// TwinCAT 3 PLC project Tc_PidControl
// ProgramVersion: 3.1.4024.0
// libraries:
//   PlantControl and CMs, * (ArmAutomation)
//   Tc2_ControllerToolbox, * (Beckhoff Automation GmbH)
//   Tc2_Standard, * (Beckhoff Automation GmbH)
//   Tc2_System, * (Beckhoff Automation GmbH)
//   Tc3_Module, * (Beckhoff Automation GmbH)
// project tree:
//   / CyclicTask100Ms.TcTTO, PlcTask.TcTTO
//   DUTs/ stParamsForScaling.TcDUT
//   GVLs/ FIO.TcGVL, GVL.TcGVL, IO.TcGVL
//   POUs/ MAIN.TcPOU
//   POUs/PID/ PRG_FB_CTRL_EmptyTank.TcPOU, PRG_FB_CTRL_PID.TcPOU, PRG_PID_CALL.TcPOU
//   POUs/Scaling/ FB_ScaleIN.TcPOU (not stored), FB_ScaleOut.TcPOU
// real-time tasks:
//   TASK PlcTask: cycle T#10ms, priority 20, ADS port 350
//   TASK CyclicTask100Ms: cycle T#100000us, priority 1, ADS port 351
// I/O:
//   DEVICE Device 1 (EtherCAT) (disabled), AmsNetId 192.168.0.244.2.1
//     Term 1 (EK1200) [EK1200-5000 EtherCAT Power supply (2A E-Bus)]
//       Term 2 (EL1008) [EL1008 8Ch. Dig. Input 24V, 3ms]
//       Term 3 (EL2008) [EL2008 8Ch. Dig. Output 24V, 0.5A]
//       Term 4 (EL3044) [EL3044 4Ch. Ana. Input 0-20mA]
//       Term 5 (EL3174) [EL3174 4Ch. Ana. Input +/-10V Diff., +/-20mA SingleEnded, 16 Bit]
//       Term 6 (EL4014) [EL4014 4Ch. Ana. Output 0-20mA, 12bit]
// variable links:
//   Tc_PidControl/Tc_PidControl Instance <-> Device 1 (EtherCAT)/Term 1 (EK1200)/Term 5 (EL3174)
//     PlcTask Inputs/IO.aiSpare02c <-> AI Standard Channel 3/Value
//     PlcTask Inputs/IO.aiSpare02d <-> AI Standard Channel 4/Value

CONFIGURATION Tc_PidControl
    RESOURCE PLC ON TwinCAT3
        TASK CyclicTask100Ms(INTERVAL := T#100000us, PRIORITY := 1);
        TASK PlcTask(INTERVAL := T#10ms, PRIORITY := 20);
        PROGRAM PRG_PID_CALL WITH CyclicTask100Ms : PRG_PID_CALL;
        PROGRAM MAIN WITH PlcTask : MAIN;
    END_RESOURCE
END_CONFIGURATION

// ---- DUTs/stParamsForScaling.TcDUT
TYPE stParamsForScaling :
STRUCT
	
    tCtrlCycleTime  : TIME := T#0ms; 
    tTaskCycleTime  : TIME := T#0ms; 
    fInMin          : REAL;
    fInMax          : REAL;
    fOutMin         : REAL;
    fOutMax         : REAL;
	
END_STRUCT

END_TYPE

// ---- GVLs/FIO.TcGVL
{attribute 'qualified_only'}
VAR_GLOBAL
	
	//	Sensor/Actuator	 Data TYPE	 Name	 Address	 Current Value
	//	Sensor	BOOL	FACTORY I/O (Running)	496	FALSE
	//	Sensor	Bool	FACTORY I/O (Paused)	497	FALSE
	//	Sensor	Bool	FACTORY I/O (Reset)	498	FALSE
	//bStart : BOOL;//	Sensor	Bool	Start	0	FALSE
	//bStop : BOOL;//	Sensor	Bool	Stop	1	TRUE
	//bReset : BOOL;//	Sensor	Bool	Reset	2	FALSE
	//	Sensor	Float	FACTORY I/O (Time Scale)	240	0
	rFlowMeter : REAL;	//	Sensor	Float	Flow meter	1	0
	rLevelMeter : REAL;	//	Sensor	Float	Level meter	0	0
	rSetPoint : REAL;	//	Sensor	Float	Setpoint	2	0
	rDisturbanceInput : REAL;
	rDisturbanceDisplay : DINT;
	//	Actuator	Bool	FACTORY I/O (Run)	496	FALSE
	//	Actuator	Bool	FACTORY I/O (Pause)	497	FALSE
	//	Actuator	Bool	FACTORY I/O (Reset)	498	FALSE
	//	Actuator	Bool	Start light	0	FALSE
	//	Actuator	Bool	Stop light	1	FALSE
	//	Actuator	Bool	Reset light	2	FALSE
	rDischargeValve : REAL;//	Actuator	Float	Discharge valve	1	0
	rFillValve : REAL;//	Actuator	Float	Fill valve	0	0
	//	Actuator	Int	FACTORY I/O (Camera Position)	240	0
	iSP : DINT;//	Actuator	Int	SP	0	0
	iPV : DINT;//	Actuator	Int	PV	1	0

END_VAR

// ---- GVLs/GVL.TcGVL
{attribute 'qualified_only'}
VAR_GLOBAL
	rAIInput1 : REAL;
	rAIInput2 : REAL;
	
	fSetpointValueToScope : LREAL;
	fActualValueToScope : LREAL;
	foutToScope : LREAL;
	
	outputDischargeValve : REAL;
	scaledDisturbancePotmeter : REAL;
	
	StartStep5 : BOOL;
	StartStep10 : BOOL;
	StartStep15 : BOOL;
	
	setManual : BOOL;
	setAuto : BOOL;
	
END_VAR

// ---- GVLs/IO.TcGVL
{attribute 'qualified_only'}
VAR_GLOBAL
	
	//EL3044
	aiSpare01a AT %I*: INT;
	aiSpare01b AT %I*: INT;
	aiSpare01c AT %I*: INT;
	aiSpare01d AT %I*: INT;
	
	//EL3074
	aiSpare02a AT %I*: INT;
	aiSpare02b AT %I*: INT;
	aiSpare02c AT %I*: INT; //ch3 0-10v  Legacy range			(0-32767)
	aiSpare02d AT %I*: INT; //ch4 0-20mA Extended range 		(0 -30518)
	
END_VAR

// ---- POUs/PID/PRG_PID_CALL.TcPOU
PROGRAM PRG_PID_CALL
VAR
	fbPlantControl : PlantAndCMs.FB_PlantControl_mode_2;
	Udt_FbPlantControl : PlantAndCMs.Udt_PlantControl_Mode_2;
	
	fbScalingSetpoint : FB_ScaleIN;
	fbScalingLevelMeter : FB_ScaleIN;
END_VAR


PRG_FB_CTRL_PID();
PRG_FB_CTRL_EmptyTank();


fbScalingSetpoint(
	taskCycletime := T#100MS,
	ctrlCycletime := T#100MS,
	inMin := 0.0,
	inMax := 10.0,
	outMin := 0.0,
	outMax := 300,
	
	inputForScaling := FIO.rSetPoint,
	
	scaledOutputInt => FIO.iSP
	);
fbScalingLevelMeter(
	taskCycletime := T#100MS,
	ctrlCycletime := T#100MS,
	inMin := 0.0,
	inMax := 10.0,
	outMin := 0.0,
	outMax := 300,
	
	inputForScaling := FIO.rLevelMeter,
	
	scaledOutputInt => FIO.iPV
	);


//aiSpare02c AT %I*: INT; //ch3 0-10v  Legacy range			(0-32767)
//measure 0-10v
//GVL.rAIInput1 := (INT_TO_REAL(IO.aiSpare02c)/(32767.0-0.0)) * 10.0;

//aiSpare02d AT %I*: INT; //ch4 0-20mA Extended range 		(0 -30518)
//measure 0-100%
//GVL.rAIInput2 := (INT_TO_REAL(IO.aiSpare02d)/(30518.0-0.0)) * 100.0;

END_PROGRAM

// ---- POUs/PID/PRG_FB_CTRL_PID.TcPOU
PROGRAM PRG_FB_CTRL_PID
VAR
	fSetpointValue					: LREAL;
	fActualValue					: LREAL;
	fManSyncValue					: LREAL;
	bSync							: BOOL;

	fOut							: LREAL;
	bHold							: BOOL;

	eMode							: E_CTRL_MODE;
	stCTRL_PID_PARAMS				: ST_CTRL_PID_PARAMS;

	eErrorId						: E_CTRL_ERRORCODES;
	bError							: BOOL;
	bARWactive						: BOOL;

	(* controller *)
	fbCTRL_PID						: FB_CTRL_PID;

	bInit							: BOOL	:= TRUE;
	fbTON							: TON;
	
	// Scaling input
	
	
	fbScalingFillValve : FB_ScaleIN;
	
	
	
END_VAR


IF GVL.setManual THEN
	eMode :=  4;	
END_IF
IF GVL.setAuto OR (GVL.StartStep5 AND GVL.StartStep10) THEN
	eMode :=  2;
ELSE
	eMode :=  0;	
END_IF



IF bInit THEN
	(* init parameter struct *)
	stCTRL_PID_PARAMS.tCtrlCycleTime		:= T#500MS;	//used to control the actual sample time of the PID algorythm, must be = or > than the task cycle time
	stCTRL_PID_PARAMS.tTaskCycleTime		:= T#100MS;		// must be the same as the cycletime configured in the task which the regulator is called in (CyclicTask100Ms)
	stCTRL_PID_PARAMS.fKp					:= 5.0;			(* proportional gain Kp				*)
	stCTRL_PID_PARAMS.tTn					:= T#100S;		(*  Tn								*)
	stCTRL_PID_PARAMS.tTv					:= T#200MS;		(*  Tv								*)
	stCTRL_PID_PARAMS.tTd					:= T#500MS;		(*  Td								*)
	stCTRL_PID_PARAMS.fOutMaxLimit			:=  100.0;			(* maximum output limit			(for  fillValve)	*) 
	stCTRL_PID_PARAMS.fOutMinLimit			:= -0.0;			(* minimum output limit			(for  fillValve)	*)

	(* set the mode to ACTIVE --> normal operation *)
	eMode := eCTRL_MODE_ACTIVE;

	(* reset the init flag *)
	bInit := FALSE;
END_IF

(*
TYPE E_CTRL_MODE :
(
    eCTRL_MODE_IDLE       := 0, (* mode idle *)
    eCTRL_MODE_PASSIVE    := 1, (* mode passive *)
    eCTRL_MODE_ACTIVE     := 2, (* mode active *)
    eCTRL_MODE_RESET      := 3, (* mode reset *)
    eCTRL_MODE_MANUAL     := 4, (* mode manual *)
    eCTRL_MODE_TUNE       := 5, (* mode tuning *)
    eCTRL_MODE_SELFTEST       := 6, (* mode selftest *)
    eCTRL_MODE_SYNC_MOVEMENT  := 7  (* mode synchronize *)
);
END_TYPE
*)

fActualValue :=  FIO.iPV; 	//FIO.rLevelMeter;
fSetpointValue := FIO.iSP; //FIO.rSetPoint (0-10V Scaled to 0-300 cm)

(* copy var to scope var *)
GVL.fSetpointValueToScope 	:= fSetpointValue;
GVL.fActualValueToScope 	:= fActualValue;


(* call controller *)
fbCTRL_PID(		fSetpointValue		:= fSetpointValue,
				fActualValue		:= fActualValue, //feedback value (proces variable)
				fManSyncValue		:= fManSyncValue, // controll fOut directly with 0-100 %?
				bSync				:= bSync,
				eMode				:= eMode,
				bHold				:= bHold,
				stParams			:= stCTRL_PID_PARAMS,
				fOut				=> fOut, // output to PID
				bARWactive			=> bARWactive,
				eErrorId			=> eErrorId,
				bError				=> bError
				);


(* copy var to scope var *)
GVL.fOutToScope := fOut;
FIO.rFillValve :=  fOut;

GVL.outputDischargeValve := fOut;




fbScalingFillValve( 
	taskCycletime := T#100MS,
	ctrlCycletime := T#100MS,
	inMin := 0.0,
	inMax := 100.0,
	outMin := 0.0,
	outMax := 10.0,
	
	inputForScaling := fOut,
	
	scaledOutputInt => FIO.rFillValve
	);

END_PROGRAM

// ---- POUs/PID/PRG_FB_CTRL_EmptyTank.TcPOU
PROGRAM PRG_FB_CTRL_EmptyTank

VAR
	fSetpointValue					: LREAL;
	fActualValue					: LREAL;
	fManSyncValue					: LREAL;
	bSync							: BOOL;

	fOut							: LREAL;
	bHold							: BOOL;

	eMode							: E_CTRL_MODE;
	stCTRL_PID_PARAMS				: ST_CTRL_PID_PARAMS;

	eErrorId						: E_CTRL_ERRORCODES;
	bError							: BOOL;
	bARWactive						: BOOL;
	
	(* controller *)
	fbCTRL_PID						: FB_CTRL_PID;
	
	bInit							: BOOL	:= TRUE;
	
	fbScalingDischargeValveInput : FB_ScaleIN;
	
	//Scaling output
	fbScalingDischargeDisturbance : FB_ScaleOut;
END_VAR

IF GVL.setManual THEN
	eMode :=  4;	
END_IF
IF GVL.setAuto AND GVL.StartStep10 THEN
	eMode :=  2;	
ELSE
	eMode :=  0;
END_IF


IF bInit THEN
	(* init parameter struct *)
	stCTRL_PID_PARAMS.tCtrlCycleTime		:= T#1000MS;	//used to control the actual sample time of the PID algorythm, must be = or > than the task cycle time
	stCTRL_PID_PARAMS.tTaskCycleTime		:= T#100MS;		// must be the same as the cycletime configured in the task which the regulator is called in (CyclicTask100Ms)
	stCTRL_PID_PARAMS.fKp					:= 5.0 ;			(* proportional gain Kp				*)
	stCTRL_PID_PARAMS.tTn					:= T#20S;		(*  Tn								*)
	stCTRL_PID_PARAMS.tTv					:= T#200MS;		(*  Tv								*)
	stCTRL_PID_PARAMS.tTd					:= T#500MS;		(*  Td								*)
	stCTRL_PID_PARAMS.fOutMaxLimit			:=  100.0;			(* maximum output limit			(for  fillValve)	*) 
	stCTRL_PID_PARAMS.fOutMinLimit			:= 0.0;			(* minimum output limit			(for  fillValve)	*)

	(* set the mode to ACTIVE --> normal operation *)
	eMode := eCTRL_MODE_ACTIVE;

	(* reset the init flag *)
	bInit := FALSE;
END_IF

fActualValue :=  FIO.iPV; 	//FIO.rLevelMeter;
fSetpointValue := FIO.iSP; //FIO.rSetPoint (0-10V Scaled to 0-300 cm)

(* call controller *)
fbCTRL_PID(		fSetpointValue		:= - 1.0 * fSetpointValue,
				fActualValue		:= -1.0 * fActualValue, //feedback value (proces variable)
				fManSyncValue		:= fManSyncValue, // controll fOut directly with 0-100 %?
				bSync				:= bSync,
				eMode				:= eMode,
				bHold				:= bHold,
				stParams			:= stCTRL_PID_PARAMS,
				fOut				=> fOut, // output to PID
				bARWactive			=> bARWactive,
				eErrorId			=> eErrorId,
				bError				=> bError
				);


(* copy var to scope var *)
//GVL.fOutToScope := fOut;
//FIO.rDischargeValve :=  fOut;

fbScalingDischargeDisturbance( 
	taskCycletime := T#100MS,
	ctrlCycletime := T#100MS,
	inMin := 0.0,
	inMax := 100.0,
	outMin := 0.0,
	outMax := 10.0,
	
	inputForScaling := fOut,
	
	scaledOutput => FIO.rDischargeValve
	);


//Manually set discharge disturbance
IF GVL.setManual THEN
	fbScalingDischargeDisturbance( 
	taskCycletime := T#100MS,
	ctrlCycletime := T#100MS,
	inMin := 0.0,
	inMax := 100.0,
	outMin := 0.0,
	outMax := 10.0,
	
	inputForScaling := FIO.rDisturbanceDisplay,
	
	scaledOutput => FIO.rDischargeValve
	);
fbScalingDischargeValveInput(
	taskCycletime := T#100MS,
	ctrlCycletime := T#100MS,
	inMin := 0.0,
	inMax := 10.0,
	outMin := 0.0,
	outMax := 100,
	
	inputForScaling := FIO.rDisturbanceInput,
	
	scaledOutputInt => FIO.rDisturbanceDisplay
	);
END_IF

END_PROGRAM

// ---- POUs/Scaling/FB_ScaleOut.TcPOU
FUNCTION_BLOCK FB_ScaleOut
VAR_INPUT
	inputForScaling : REAL;
	inMin : REAL;
	inMax : REAL;
	outMin : REAL;
	outMax : REAL;
	ctrlCycletime : TIME;
	taskCycletime : TIME;
END_VAR
VAR_OUTPUT
	scaledOutput : real;
END_VAR
VAR
	fbScale : FB_CTRL_SCALE;
	stParamsForScaling : ST_CTRL_SCALE_PARAMS;
	
END_VAR

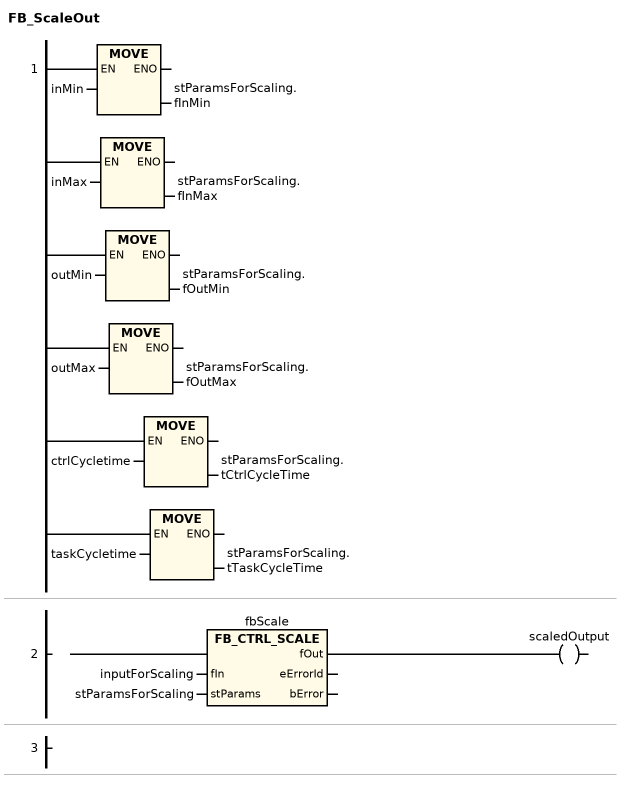
// NETWORK 1
stParamsForScaling.fInMin := inMin;
stParamsForScaling.fInMax := inMax;
stParamsForScaling.fOutMin := outMin;
stParamsForScaling.fOutMax := outMax;
stParamsForScaling.tCtrlCycleTime := ctrlCycletime;
stParamsForScaling.tTaskCycleTime := taskCycletime;

// NETWORK 2
fbScale(fIn := inputForScaling, stParams := stParamsForScaling); // FB_CTRL_SCALE
scaledOutput := fbScale.fOut;

// NETWORK 3

END_FUNCTION_BLOCK

// ---- POUs/MAIN.TcPOU
PROGRAM MAIN
VAR
	fbPlantControl : PlantAndCMs.FB_PlantControl_mode_1;
	Udt_FbPlantControl : PlantAndCMs.Udt_PlantControl_Mode_1;
	
	testCase_step : INT := 0;
	
	Timer_Step10 : TON;
END_VAR

Timer_Step10(IN:= , PT:= T#50S, Q=> , ET=> );

fbPlantControl(
	Start_In := PlantAndCMs.FIO.bStart,
	Stop_In := PlantAndCMs.FIO.bStop, 
	Reset_In := PlantAndCMs.FIO.bReset,
	EmgStop_In := PlantAndCMs.FIO.bEmgStop,
	
	Auto_In := PlantAndCMs.FIO.bAuto,
	Manual_In := PlantAndCMs.FIO.bManual,
	
	Ctrl_Plant := Udt_FbPlantControl
	);

IF fbPlantControl.Manual_Out AND NOT fbPlantControl.Auto_Out THEN
	GVL.setManual := TRUE;
	GVL.setAuto := FALSE;
ELSE
	GVL.setManual := FALSE;
	GVL.setAuto := TRUE;
END_IF

	
CASE testCase_step OF
	0: // init:
	
	IF fbPlantControl.Auto_Out THEN
		testCase_step := 1;
	END_IF
	
	1:
	IF fbPlantControl.Startet_Out THEN
		testCase_step := 5;
	END_IF
	
	5: // fill tank up to setpoint 100
	GVL.StartStep5 := TRUE;
	FIO.iSP := 100;
	
	IF FIO.iPV = 100 THEN
		GVL.StartStep5 := FALSE;
		testCase_step := 10;
	END_IF
	
	10: // empty tank to set point 50
	GVL.StartStep10 := TRUE;
	Timer_Step10.IN := TRUE;
	
	FIO.iSP := 25;
	
	IF  Timer_Step10.Q THEN
		testCase_step := 15;
	END_IF
	
	15:
	
	IF FIO.iPV = 25 THEN
		testCase_step := 5;
	END_IF
	
	
END_CASE

END_PROGRAM
